(* CoDeSys 2.3 export: FX_PORTEG.EXP *)

(* POU Simulation_Visuelle/FX_PorteG, ST *)
FUNCTION FX_PorteG : REAL
VAR_INPUT
	PosXPorte: REAL;
END_VAR
VAR
	VarLocalA: REAL;
END_VAR
(*Cette fonction retourne la position Y en fonction de l'axe X de la porte gauche*)
VarLocalA:=(20.0/59.0);
VarLocalA:=(VarLocalA)*(PosXPorte);
FX_PorteG:=VarLocalA +1;
END_FUNCTION
